FUNCTION_BLOCK TankFuellAnlage
VAR_INPUT
END_VAR
VAR_OUTPUT
END_VAR
VAR
END_VAR

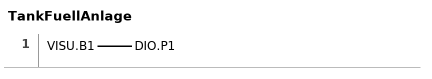
// NETWORK 1
DIO.P1 := VISU.B1;

END_FUNCTION_BLOCK

(* stored: Version 1.1.0.1, ProductVersion 3.1.4022.6
   POU TankFuellAnlage: Id {d266dc57-a678-43a7-8e11-96d978017ed9}, SpecialFunc None *)
